FUNCTION_BLOCK FB_State1 EXTENDS FB_State
VAR_INPUT
END_VAR
VAR_OUTPUT
END_VAR
VAR
END_VAR

END_FUNCTION_BLOCK

(* stored: Version 1.1.0.1, ProductVersion 3.1.4024.12
   POU FB_State1: Id {915978e7-92ee-4f02-a74f-b5db3f8bd174}, SpecialFunc None *)
